# EPICS substitutions: apps/mmfeuApp/Db/mmfeusumsFTT.substitutions
file "db/mmfeusumsFTT.db" {
pattern { SUFFIX }
{ Current_A }
{ XTmpV6_deg }
{ MTmpInt_deg }
{ TmpSdX_deg }
{ TmpSdA_deg }
}
